TYPE ST_StationTrackPosition :
STRUCT
	fPositionOnTrack	: LREAL;
	nTrackId			: INT;	
END_STRUCT
END_TYPE

(* stored: Version 1.1.0.1, ProductVersion 3.1.4024.9
   DUT ST_StationTrackPosition: Id {da0f2790-38c7-4db6-bd89-b5280a607df3} *)
